{attribute 'qualified_only'}
{attribute 'strict'}
TYPE E_StationProcessState :
(
	Idle 			:= 0,
	ProcessStart 	:= 1,
	ProcessBusy 	:= 2,
	ProcessDone 	:= 3
);
END_TYPE

(* stored: Version 1.1.0.1, ProductVersion 3.1.4024.12
   DUT E_StationProcessState: Id {644be6a6-2762-46c6-b2b0-5797d19cb43b} *)
